// TIA Portal V16 export
// export: Created 2023-03-29T11:04:56.9230483Z, ExportSetting WithDefaults, DisplayName Totally Integrated Automation Portal, DisplayVersion V16 Update 6, DisplayName TIA Portal Version Control Interface, DisplayVersion V16 Update 2, DisplayName TIA Portal Openness, DisplayVersion V16 Update 6, DisplayName STEP 7 Professional, DisplayVersion V16 Update 6, DisplayName STEP 7 Safety, DisplayVersion V16, DisplayName WinCC Advanced, DisplayVersion V16 Update 6
DATA_BLOCK "dbControll modors leading and extras"   // DB46
AUTHOR : rtecmer
VERSION : 0.1
// stored: AutoNumber true, DBAccessibleFromOPCUA true, InstanceOfName Ustawienie pomp wiodącej i dodatkowych, InstanceOfType FB
"Ustawienie pomp wiodącej i dodatkowych"
   // VAR_IN_OUT
   //    set_Motor2 : Bool;
   //    set_Motor3 : Bool;
   //    set_Motor4 : Bool;
   // END_VAR
BEGIN
END_DATA_BLOCK
